FUNCTION_BLOCK FB_LamparaComputada_SFC
VAR_INPUT
    ReiniciaContador: BOOL;
    ManiobrasTotales: UINT := 2;
    TiempoEncendido: REAL := 2.0;
END_VAR
VAR_OUTPUT
    LamparaHabilitada: BOOL;
    ManiobrasPendientes: UINT := ManiobrasTotales;
    TiempoPendiente: REAL;
END_VAR
VAR
    Lampara AT %Q*: BOOL;
    Pulsador AT %I*: BOOL;
END_VAR

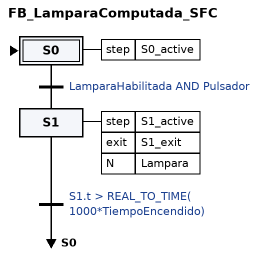
INITIAL_STEP S0:
    S0_active(N);  // step action
END_STEP
TRANSITION FROM S0 TO S1
    := LamparaHabilitada AND Pulsador;
END_TRANSITION
STEP S1:
    S1_active(N);  // step action
    S1_exit(P0);  // exit action
    Lampara(N);
END_STEP
TRANSITION FROM S1 TO S0
    := S1.t > REAL_TO_TIME(1000*TiempoEncendido);
END_TRANSITION

ACTION S0_active:
LamparaHabilitada := (ManiobrasPendientes > 0);

IF ReiniciaContador THEN 
    ManiobrasPendientes := ManiobrasTotales;
END_IF
END_ACTION

ACTION S1_active:
TiempoPendiente := TiempoEncendido - (TIME_TO_REAL(S1.t)/1000);
END_ACTION

ACTION S1_exit:
IF (ManiobrasPendientes > 0) THEN 
    ManiobrasPendientes := ManiobrasPendientes - 1;
END_IF
END_ACTION

END_FUNCTION_BLOCK

(* stored: Version 1.1.0.1, ProductVersion 3.1.4024.15
   POU FB_LamparaComputada_SFC: Id {5017c17c-8705-42a3-821d-8ab471c59e55}, SpecialFunc None
   Action S0_active: Id {2e47c035-9f95-4cbc-94d9-bf2b2c727cb0}
   Action S1_active: Id {e8a42836-b0a7-434d-b652-4e5ec8b982ff}
   Action S1_exit: Id {290c5996-f693-446c-9961-0761e0f5c222} *)
